// TIA Portal V16 export
// export: Created 2023-03-29T11:05:03.6986651Z, ExportSetting WithDefaults, DisplayName Totally Integrated Automation Portal, DisplayVersion V16 Update 6, DisplayName TIA Portal Version Control Interface, DisplayVersion V16 Update 2, DisplayName TIA Portal Openness, DisplayVersion V16 Update 6, DisplayName STEP 7 Professional, DisplayVersion V16 Update 6, DisplayName STEP 7 Safety, DisplayVersion V16, DisplayName WinCC Advanced, DisplayVersion V16 Update 6
VAR_GLOBAL   // PLC tag table "PID"
   switc_manualPID AT %M206.5 : Bool;   // Przełacznik regulator PID na manualne zadawanie
   setUP_O2 AT %M300.3 : Bool;   // Znacznik generatora czasowego podnoszenia wartości zadanej ciśnienia
   setDown_O2 AT %M300.4 : Bool;   // Znacznik generatora czasowego obniżania wartości ciśnienia
END_VAR
